FUNCTION_BLOCK FB_Hmi_Button
VAR
	_rButton: REFERENCE TO S_Hmi_Button;

	_Led: FB_Hmi_Led;

	_behaviour: E_Hmi_ButtonBehaviour;
	_value: BOOL;

	_initialized: BOOL;
END_VAR

IF _initialized THEN
	IF _behaviour = E_Hmi_ButtonBehaviour.MomentaryOff THEN
		_value := TRUE;
	ELSIF _behaviour = E_Hmi_ButtonBehaviour.MomentaryOn THEN
		_value := FALSE;
	END_IF

	IF _rButton.Click THEN
		CASE _behaviour OF
			E_Hmi_ButtonBehaviour.MomentaryOff:
				Reset();

			E_Hmi_ButtonBehaviour.MomentaryOn:
				Set();

			E_Hmi_ButtonBehaviour.Reset:
				Reset();

			E_Hmi_ButtonBehaviour.Set:
				Set();

			E_Hmi_ButtonBehaviour.Toggle:
				Toggle();
		END_CASE

		_rButton.Click := FALSE;
	END_IF
END_IF

PROPERTY PUBLIC Enabled : BOOL
SET
_rButton.Enabled := Enabled;
END_SET
END_PROPERTY

METHOD PUBLIC Initialize : BOOL
VAR_INPUT
	rButton: REFERENCE TO S_Hmi_Button;
	behaviour: E_Hmi_ButtonBehaviour;
END_VAR
IF __ISVALIDREF(rButton) THEN
	_Led.initialize(rButton.Led);
	_rButton REF= rButton;
	_behaviour := behaviour;

	_initialized := Initialize := TRUE;
END_IF
END_METHOD

PROPERTY PUBLIC Led : POINTER TO FB_Hmi_Led;
GET
Led := ADR(_Led);
END_GET
END_PROPERTY

METHOD PUBLIC Reset
IF _initialized AND_THEN _rButton.Enabled THEN
	_value := FALSE;
END_IF
END_METHOD

METHOD PUBLIC Set
IF _initialized AND_THEN _rButton.Enabled THEN
	_value := TRUE;
END_IF
END_METHOD

METHOD PUBLIC Toggle
IF _initialized AND_THEN _rButton.Enabled THEN
	_value := NOT _value;
END_IF
END_METHOD

PROPERTY PUBLIC Value : BOOL
GET
Value := _value;
END_GET
END_PROPERTY

PROPERTY PUBLIC Visibility : BOOL
SET
IF _initialized THEN
	_rButton.Visibility := Visibility;
END_IF
END_SET
END_PROPERTY

END_FUNCTION_BLOCK

(* stored: Version 1.1.0.1, ProductVersion 3.1.4024.10
   POU FB_Hmi_Button: Id {a617f7ad-fb3b-4a46-851f-875681a96aba}, SpecialFunc None
   Property Enabled: Id {5b4cf018-ce66-4b92-8000-7260fe469dc8}
   Set Set: Id {2793329d-7047-48a2-9868-24a2d32378e8}
   Method Initialize: Id {e3910462-5f99-46e6-a6aa-9b16848dc198}
   Property Led: Id {2886d8f7-91ae-4509-a03a-8ce26d6320e8}
   Get Get: Id {d00133b7-c570-4520-9dd4-1cc0b8ddc711}
   Method Reset: Id {e5c166a3-5f3c-4eb9-b57a-708a2a6197b7}
   Method Set: Id {d110b873-8a6f-4d1f-b710-60c6a34d74e5}
   Method Toggle: Id {2e7dfe79-cc01-47d2-a514-773e8cd4ab1d}
   Property Value: Id {4699e93b-d29c-4866-a3a4-a35fe790999d}
   Get Get: Id {ba3d2ae5-2beb-480e-86ae-d9f4f4c013ab}
   Property Visibility: Id {f2b03956-52c9-4261-87db-41fea13bbf68}
   Set Set: Id {ec4b2845-fad5-44c3-a7ee-34244c9bb334} *)
